# EPICS alarm handler configuration: mps_database/bareTest/alarms/areas/mpln_bpn26_mp01.alhConfig
GROUP NULL MPLN:BPN26:MP01:1
$ALIAS MPS Link Node 90
$GUIDANCE
LTUH MPS
   Group Name: MPLN:BPN26:MP01:1
   Summary PV:  MPLN:BPN26:MP01:1:STATSUMY
$END
CHANNEL  MPLN:BPN26:MP01:1    MPLN:BPN26:MP01:1:MPS_EN_RBV		-----
CHANNEL  MPLN:BPN26:MP01:1    MPLN:BPN26:MP01:1:LC1_MODE_RBV		-----
